ABB RobotStudio station: kostka_final.rspag

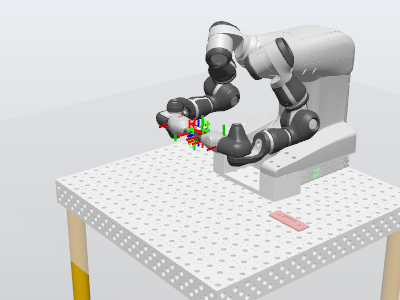
--- station ---
Station kostka (saved by RobotStudio 24.1.10693.0)
Controller Controller1
  mechanical unit ROB_R: IRB14000_0.5_0.5_R, 6 joints, base frame (0, 0, 0) mm
  mechanical unit ROB_R_7: IRB14000_0.5_0.5_R, 1 joints, base frame (0, 0, 0) mm
  mechanical unit ROB_L: IRB14000_0.5_0.5_L, 6 joints, base frame (0, 0, 0) mm
  mechanical unit ROB_L_7: IRB14000_0.5_0.5_L, 1 joints, base frame (0, 0, 0) mm
Layout (positions relative to the parent item):
  - Workplace [part, from Components\Table_for_yumi.rslib] at (-401.98, -347.06, -251) mm
  - IRB14000_0.5_0.5 [mechanism, from %ABB.RobotStudio.Models.IRB14000%\IRB14000_0.5_0.5__02.rslib] at (0, 0, 0) mm
  - IRB14000_0.5_0.5_R [mechanism, from %ABB.RobotStudio.Models.IRB14000%\IRB14000_0.5_0.5__02.rslib] at (0, 0, 0) mm; joint values [1.5163, -2.3974, -0.8514, 0.598, -1.3187, 1.4925, 3.1384] (rad or m)
  - IRB14000_0.5_0.5_L [mechanism, from %ABB.RobotStudio.Models.IRB14000%\IRB14000_0.5_0.5__02.rslib] at (0, 0, 0) mm; joint values [-1.536, -2.4067, 0.8768, 0.6099, 1.3554, 1.4655, 3.1349] (rad or m)
  - Smart_Gripper_Servo_Fingers_R [mechanism] at (341.28, 130.02, 173.54) mm, rotated rx 90 ry 0 rz 0 deg; joint values [0.023] (rad or m)
      TCP Servo at (0, 0, 114.2) mm
      links: HandBase, DownFinger, UpFinger, VacuumOne, VacuumTwo
  - Smart_Gripper_Servo_Fingers_2L [mechanism] at (341.28, -144.48, 173.54) mm, rotated rx -90 ry 0 rz 0 deg; joint values [0.023] (rad or m)
      TCP Servo at (0, 0, 114.2) mm
      links: HandBase, DownFinger, UpFinger, VacuumOne, VacuumTwo
  - Node1_con [part] at (329.77, -18.73, 185.04) mm, size 23 x 23 x 23 mm
  - Node2_con [part] at (329.77, 4.27, 162.04) mm, size 23 x 23 x 23 mm
  - Node3_con [part] at (352.77, 4.27, 162.04) mm, size 23 x 23 x 23 mm
  - Node4_con [part] at (329.78, -18.73, 162.04) mm, size 23 x 23 x 23 mm
  - Node5_con [part] at (352.77, -18.73, 162.04) mm, size 23 x 23 x 23 mm
  - Node6_con [part] at (352.77, 4.27, 185.04) mm, size 23 x 23 x 23 mm
  - Node7_con [part] at (329.77, 4.27, 185.04) mm, size 23 x 23 x 23 mm
  - Node8_con [part] at (352.77, -18.73, 185.04) mm, size 23 x 23 x 23 mm
  - Positioner [smart component, from Components\Positioner.rslib]
      properties: Object=Node1_con; Position=[0.329775 -0.01873 0.185036]; Orientation=[0 0 0]; Reference=Global; ReferenceObject=(none)
  - Positioner_2 [smart component, from Components\Positioner.rslib]
      properties: Object=Node2_con; Position=[0.329775 0.00427 0.162037]; Orientation=[0 0 0]; Reference=Global; ReferenceObject=(none)
  - Positioner_3 [smart component, from Components\Positioner.rslib]
      properties: Object=Node3_con; Position=[0.352771 0.00427 0.162036]; Orientation=[0 0 0]; Reference=Global; ReferenceObject=(none)
  - Positioner_4 [smart component, from Components\Positioner.rslib]
      properties: Object=Node4_con; Position=[0.329775 -0.01873 0.162037]; Orientation=[0 0 0]; Reference=Global; ReferenceObject=(none)
  - Positioner_5 [smart component, from Components\Positioner.rslib]
      properties: Object=Node5_con; Position=[0.352771 -0.01873 0.162036]; Orientation=[0 0 0]; Reference=Global; ReferenceObject=(none)
  - Positioner_6 [smart component, from Components\Positioner.rslib]
      properties: Object=Node6_con; Position=[0.352771 0.00427 0.185036]; Orientation=[0 0 0]; Reference=Global; ReferenceObject=(none)
  - Positioner_7 [smart component, from Components\Positioner.rslib]
      properties: Object=Node7_con; Position=[0.329775 0.00427 0.185036]; Orientation=[0 0 0]; Reference=Global; ReferenceObject=(none)
  - Positioner_8 [smart component, from Components\Positioner.rslib]
      properties: Object=Node8_con; Position=[0.352771 -0.01873 0.185036]; Orientation=[0 0 0]; Reference=Global; ReferenceObject=(none)
Attachment: Smart_Gripper_Servo_Fingers_R is attached to IRB14000_0.5_0.5_L / Link7
Attachment: Smart_Gripper_Servo_Fingers_2L is attached to IRB14000_0.5_0.5_R / Link7
Attachment: Node6_con is attached to Smart_Gripper_Servo_Fingers_R / HandBase
Attachment: Node7_con is attached to Smart_Gripper_Servo_Fingers_R / HandBase
Attachment: Node3_con is attached to Smart_Gripper_Servo_Fingers_R / HandBase
Attachment: Node2_con is attached to Smart_Gripper_Servo_Fingers_R / HandBase
Attachment: Node8_con is attached to Smart_Gripper_Servo_Fingers_2L / HandBase
Attachment: Node1_con is attached to Smart_Gripper_Servo_Fingers_2L / HandBase
Attachment: Node4_con is attached to Smart_Gripper_Servo_Fingers_2L / HandBase
Attachment: Node5_con is attached to Smart_Gripper_Servo_Fingers_2L / HandBase
EventTableEntry 7537: ActivationMode=2, Cyclic=false, Group=, Trigger=DO_ATTACH_1_GL 7538, Actions=[EventTableActionAttach 7572, EventTableActionAttach 7573, EventTableActionAttach 7574, EventTableActionAttach 7575], Comment=
EventTableTriggerIO 7538: Operator=0, IOValue=[1], IRC5Controller=? -1, SignalSource=Controller1 3578
EventTableEntry 7543: ActivationMode=2, Cyclic=false, Group=, Trigger=DO_DETACH_GL 7544, Actions=[EventTableActionDetach 7545], Comment=
EventTableTriggerIO 7544: Operator=0, IOValue=[1], IRC5Controller=? -1, SignalSource=Controller1 3578
EventTableActionDetach 7545: AttachmentParent=Smart_Gripper_Servo_Fingers_2L 3564, AttachmentChild=? -1
EventTableTriggerIO 7564: Operator=0, IOValue=[1], IRC5Controller=? -1, SignalSource=Controller1 3578
EventTableTriggerIO 7565: Operator=0, IOValue=[1], IRC5Controller=? -1, SignalSource=Controller1 3578
EventTableTriggerIO 7566: Operator=0, IOValue=[1], IRC5Controller=? -1, SignalSource=Controller1 3578
EventTableTriggerIO 7567: Operator=0, IOValue=[1], IRC5Controller=? -1, SignalSource=Controller1 3578
EventTableTriggerIO 7568: Operator=0, IOValue=[1], IRC5Controller=? -1, SignalSource=Controller1 3578
EventTableTriggerIO 7569: Operator=0, IOValue=[1], IRC5Controller=? -1, SignalSource=Controller1 3578
EventTableTriggerIO 7570: Operator=0, IOValue=[1], IRC5Controller=? -1, SignalSource=Controller1 3578
EventTableTriggerIO 7571: Operator=0, IOValue=[1], IRC5Controller=? -1, SignalSource=Controller1 3578
EventTableActionAttach 7572: MountObject=false, FlangeIndext=0, FindNearest=false, AttachmentParent=Smart_Gripper_Servo_Fingers_2L 3564, AttachmentChild=Node8_con 7749, Offset=[X=1, Y=0, Z=0, W=0, X=0, Y=1, Z=0, W=0, X=0, Y=0, Z=1, W=0, X=0, Y=0, Z=0, W=1]
EventTableActionAttach 7573: MountObject=false, FlangeIndext=0, FindNearest=false, AttachmentParent=Smart_Gripper_Servo_Fingers_2L 3564, AttachmentChild=Node6_con 7745, Offset=[X=1, Y=0, Z=0, W=0, X=0, Y=1, Z=0, W=0, X=0, Y=0, Z=1, W=0, X=0, Y=0, Z=0, W=1]
EventTableActionAttach 7574: MountObject=false, FlangeIndext=0, FindNearest=false, AttachmentParent=Smart_Gripper_Servo_Fingers_2L 3564, AttachmentChild=Node5_con 7743, Offset=[X=1, Y=0, Z=0, W=0, X=0, Y=1, Z=0, W=0, X=0, Y=0, Z=1, W=0, X=0, Y=0, Z=0, W=1]
EventTableActionAttach 7575: MountObject=false, FlangeIndext=0, FindNearest=false, AttachmentParent=Smart_Gripper_Servo_Fingers_2L 3564, AttachmentChild=Node3_con 7739, Offset=[X=1, Y=0, Z=0, W=0, X=0, Y=1, Z=0, W=0, X=0, Y=0, Z=1, W=0, X=0, Y=0, Z=0, W=1]
EventTableTriggerIO 7576: Operator=0, IOValue=[1], IRC5Controller=? -1, SignalSource=Controller1 3578
EventTableEntry 7577: ActivationMode=2, Cyclic=false, Group=, Trigger=DO_ATTACH_2_GL 7564, Actions=[EventTableActionAttach 7578, EventTableActionAttach 7579, EventTableActionAttach 7580, EventTableActionAttach 7581], Comment=
EventTableActionAttach 7578: MountObject=false, FlangeIndext=0, FindNearest=false, AttachmentParent=Smart_Gripper_Servo_Fingers_2L 3564, AttachmentChild=Node8_con 7749, Offset=[X=1, Y=0, Z=0, W=0, X=0, Y=1, Z=0, W=0, X=0, Y=0, Z=1, W=0, X=0, Y=0, Z=0, W=1]
EventTableActionAttach 7579: MountObject=false, FlangeIndext=0, FindNearest=false, AttachmentParent=Smart_Gripper_Servo_Fingers_2L 3564, AttachmentChild=Node1_con 7735, Offset=[X=1, Y=0, Z=0, W=0, X=0, Y=1, Z=0, W=0, X=0, Y=0, Z=1, W=0, X=0, Y=0, Z=0, W=1]
EventTableActionAttach 7580: MountObject=false, FlangeIndext=0, FindNearest=false, AttachmentParent=Smart_Gripper_Servo_Fingers_2L 3564, AttachmentChild=Node4_con 7741, Offset=[X=1, Y=0, Z=0, W=0, X=0, Y=1, Z=0, W=0, X=0, Y=0, Z=1, W=0, X=0, Y=0, Z=0, W=1]
EventTableActionAttach 7581: MountObject=false, FlangeIndext=0, FindNearest=false, AttachmentParent=Smart_Gripper_Servo_Fingers_2L 3564, AttachmentChild=Node5_con 7743, Offset=[X=1, Y=0, Z=0, W=0, X=0, Y=1, Z=0, W=0, X=0, Y=0, Z=1, W=0, X=0, Y=0, Z=0, W=1]
EventTableEntry 7582: ActivationMode=2, Cyclic=false, Group=, Trigger=DO_ATTACH_5_GR 7568, Actions=[EventTableActionAttach 7583, EventTableActionAttach 7584, EventTableActionAttach 7585, EventTableActionAttach 7586], Comment=
EventTableActionAttach 7583: MountObject=false, FlangeIndext=0, FindNearest=false, AttachmentParent=Smart_Gripper_Servo_Fingers_R 3556, AttachmentChild=Node1_con 7735, Offset=[X=1, Y=0, Z=0, W=0, X=0, Y=1, Z=0, W=0, X=0, Y=0, Z=1, W=0, X=0, Y=0, Z=0, W=1]
EventTableActionAttach 7584: MountObject=false, FlangeIndext=0, FindNearest=false, AttachmentParent=Smart_Gripper_Servo_Fingers_R 3556, AttachmentChild=Node2_con 7737, Offset=[X=1, Y=0, Z=0, W=0, X=0, Y=1, Z=0, W=0, X=0, Y=0, Z=1, W=0, X=0, Y=0, Z=0, W=1]
EventTableActionAttach 7585: MountObject=false, FlangeIndext=0, FindNearest=false, AttachmentParent=Smart_Gripper_Servo_Fingers_R 3556, AttachmentChild=Node7_con 7747, Offset=[X=1, Y=0, Z=0, W=0, X=0, Y=1, Z=0, W=0, X=0, Y=0, Z=1, W=0, X=0, Y=0, Z=0, W=1]
EventTableActionAttach 7586: MountObject=false, FlangeIndext=0, FindNearest=false, AttachmentParent=Smart_Gripper_Servo_Fingers_R 3556, AttachmentChild=Node4_con 7741, Offset=[X=1, Y=0, Z=0, W=0, X=0, Y=1, Z=0, W=0, X=0, Y=0, Z=1, W=0, X=0, Y=0, Z=0, W=1]
EventTableEntry 7587: ActivationMode=2, Cyclic=false, Group=, Trigger=DO_DETACH_GR 7576, Actions=[EventTableActionDetach 7588], Comment=
EventTableActionDetach 7588: AttachmentParent=Smart_Gripper_Servo_Fingers_R 3556, AttachmentChild=? -1
EventTableEntry 7589: ActivationMode=2, Cyclic=false, Group=, Trigger=DO_ATTACH_4_GR 7569, Actions=[EventTableActionAttach 7590, EventTableActionAttach 7591, EventTableActionAttach 7592, EventTableActionAttach 7593], Comment=
EventTableActionAttach 7590: MountObject=false, FlangeIndext=0, FindNearest=false, AttachmentParent=Smart_Gripper_Servo_Fingers_R 3556, AttachmentChild=Node6_con 7745, Offset=[X=1, Y=0, Z=0, W=0, X=0, Y=1, Z=0, W=0, X=0, Y=0, Z=1, W=0, X=0, Y=0, Z=0, W=1]
EventTableActionAttach 7591: MountObject=false, FlangeIndext=0, FindNearest=false, AttachmentParent=Smart_Gripper_Servo_Fingers_R 3556, AttachmentChild=Node7_con 7747, Offset=[X=1, Y=0, Z=0, W=0, X=0, Y=1, Z=0, W=0, X=0, Y=0, Z=1, W=0, X=0, Y=0, Z=0, W=1]
EventTableActionAttach 7592: MountObject=false, FlangeIndext=0, FindNearest=false, AttachmentParent=Smart_Gripper_Servo_Fingers_R 3556, AttachmentChild=Node3_con 7739, Offset=[X=1, Y=0, Z=0, W=0, X=0, Y=1, Z=0, W=0, X=0, Y=0, Z=1, W=0, X=0, Y=0, Z=0, W=1]
EventTableActionAttach 7593: MountObject=false, FlangeIndext=0, FindNearest=false, AttachmentParent=Smart_Gripper_Servo_Fingers_R 3556, AttachmentChild=Node2_con 7737, Offset=[X=1, Y=0, Z=0, W=0, X=0, Y=1, Z=0, W=0, X=0, Y=0, Z=1, W=0, X=0, Y=0, Z=0, W=1]
EventTableEntry 7594: ActivationMode=2, Cyclic=false, Group=, Trigger=DO_ATTACH_3_GR 7570, Actions=[EventTableActionAttach 7595, EventTableActionAttach 7596, EventTableActionAttach 7597, EventTableActionAttach 7598], Comment=
EventTableActionAttach 7595: MountObject=false, FlangeIndext=0, FindNearest=false, AttachmentParent=Smart_Gripper_Servo_Fingers_R 3556, AttachmentChild=Node2_con 7737, Offset=[X=1, Y=0, Z=0, W=0, X=0, Y=1, Z=0, W=0, X=0, Y=0, Z=1, W=0, X=0, Y=0, Z=0, W=1]
EventTableActionAttach 7596: MountObject=false, FlangeIndext=0, FindNearest=false, AttachmentParent=Smart_Gripper_Servo_Fingers_R 3556, AttachmentChild=Node3_con 7739, Offset=[X=1, Y=0, Z=0, W=0, X=0, Y=1, Z=0, W=0, X=0, Y=0, Z=1, W=0, X=0, Y=0, Z=0, W=1]
EventTableActionAttach 7597: MountObject=false, FlangeIndext=0, FindNearest=false, AttachmentParent=Smart_Gripper_Servo_Fingers_R 3556, AttachmentChild=Node4_con 7741, Offset=[X=1, Y=0, Z=0, W=0, X=0, Y=1, Z=0, W=0, X=0, Y=0, Z=1, W=0, X=0, Y=0, Z=0, W=1]
EventTableActionAttach 7598: MountObject=false, FlangeIndext=0, FindNearest=false, AttachmentParent=Smart_Gripper_Servo_Fingers_R 3556, AttachmentChild=Node5_con 7743, Offset=[X=1, Y=0, Z=0, W=0, X=0, Y=1, Z=0, W=0, X=0, Y=0, Z=1, W=0, X=0, Y=0, Z=0, W=1]
EventTableEntry 7599: ActivationMode=2, Cyclic=false, Group=, Trigger=DO_ATTACH_6_GL 7571, Actions=[EventTableActionAttach 7600, EventTableActionAttach 7601, EventTableActionAttach 7602, EventTableActionAttach 7603], Comment=
EventTableActionAttach 7600: MountObject=false, FlangeIndext=0, FindNearest=false, AttachmentParent=Smart_Gripper_Servo_Fingers_2L 3564, AttachmentChild=Node1_con 7735, Offset=[X=1, Y=0, Z=0, W=0, X=0, Y=1, Z=0, W=0, X=0, Y=0, Z=1, W=0, X=0, Y=0, Z=0, W=1]
EventTableActionAttach 7601: MountObject=false, FlangeIndext=0, FindNearest=false, AttachmentParent=Smart_Gripper_Servo_Fingers_2L 3564, AttachmentChild=Node8_con 7749, Offset=[X=1, Y=0, Z=0, W=0, X=0, Y=1, Z=0, W=0, X=0, Y=0, Z=1, W=0, X=0, Y=0, Z=0, W=1]
EventTableActionAttach 7602: MountObject=false, FlangeIndext=0, FindNearest=false, AttachmentParent=Smart_Gripper_Servo_Fingers_2L 3564, AttachmentChild=Node7_con 7747, Offset=[X=1, Y=0, Z=0, W=0, X=0, Y=1, Z=0, W=0, X=0, Y=0, Z=1, W=0, X=0, Y=0, Z=0, W=1]
EventTableActionAttach 7603: MountObject=false, FlangeIndext=0, FindNearest=false, AttachmentParent=Smart_Gripper_Servo_Fingers_2L 3564, AttachmentChild=Node6_con 7745, Offset=[X=1, Y=0, Z=0, W=0, X=0, Y=1, Z=0, W=0, X=0, Y=0, Z=1, W=0, X=0, Y=0, Z=0, W=1]
EventTableEntry 7630: ActivationMode=2, Cyclic=false, Group=, Trigger=DO_CLOSE_GL 7631, Actions=[EventTableActionMechanicalPose 7632], Comment=
EventTableTriggerIO 7631: Operator=0, IOValue=[1], IRC5Controller=? -1, SignalSource=Controller1 3578
EventTableActionMechanicalPose 7632: VirtualSignal=, Mechanism=Smart_Gripper_Servo_Fingers_2L 3564, ToPoseName=SyncPosition, VirtualSignalValue=[1]
EventTableTriggerIO 7633: Operator=0, IOValue=[1], IRC5Controller=? -1, SignalSource=Controller1 3578
EventTableTriggerIO 7634: Operator=0, IOValue=[1], IRC5Controller=? -1, SignalSource=Controller1 3578
EventTableTriggerIO 7635: Operator=0, IOValue=[1], IRC5Controller=? -1, SignalSource=Controller1 3578
EventTableEntry 7636: ActivationMode=2, Cyclic=false, Group=, Trigger=DO_OPEN_GL 7633, Actions=[EventTableActionMechanicalPose 7637], Comment=
EventTableActionMechanicalPose 7637: VirtualSignal=, Mechanism=Smart_Gripper_Servo_Fingers_2L 3564, ToPoseName=HomePosition, VirtualSignalValue=[1]
EventTableEntry 7638: ActivationMode=2, Cyclic=false, Group=, Trigger=DO_CLOSE_GR 7634, Actions=[EventTableActionMechanicalPose 7639], Comment=
EventTableActionMechanicalPose 7639: VirtualSignal=, Mechanism=Smart_Gripper_Servo_Fingers_R 3556, ToPoseName=SyncPosition, VirtualSignalValue=[1]
EventTableEntry 7640: ActivationMode=2, Cyclic=false, Group=, Trigger=DO_OPEN_GR 7635, Actions=[EventTableActionMechanicalPose 7641], Comment=
EventTableActionMechanicalPose 7641: VirtualSignal=, Mechanism=Smart_Gripper_Servo_Fingers_R 3556, ToPoseName=HomePosition, VirtualSignalValue=[1]
EventTableTriggerIO 7692: Operator=0, IOValue=[1], IRC5Controller=? -1, SignalSource=Controller1 3578
EventTableTriggerIO 7693: Operator=0, IOValue=[1], IRC5Controller=? -1, SignalSource=Controller1 3578
EventTableTriggerIO 7694: Operator=0, IOValue=[1], IRC5Controller=? -1, SignalSource=Controller1 3578
EventTableTriggerIO 7695: Operator=0, IOValue=[1], IRC5Controller=? -1, SignalSource=Controller1 3578
EventTableTriggerIO 7696: Operator=0, IOValue=[1], IRC5Controller=? -1, SignalSource=Controller1 3578
EventTableTriggerIO 7697: Operator=0, IOValue=[1], IRC5Controller=? -1, SignalSource=Controller1 3578
EventTableTriggerIO 7698: Operator=0, IOValue=[1], IRC5Controller=? -1, SignalSource=Controller1 3578
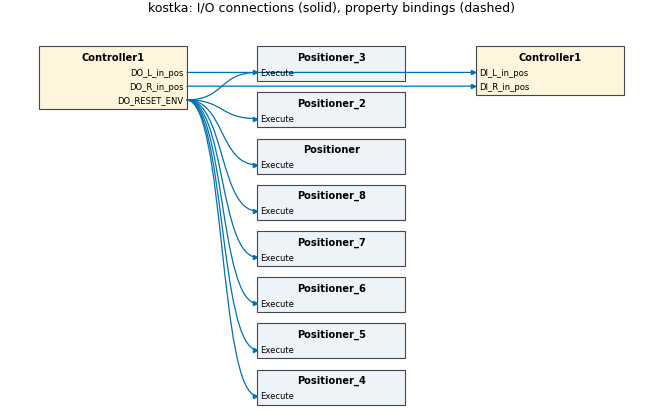
Station logic (signal -> signal, property => property):
  Controller1.DO_L_in_pos -> Controller1.DI_L_in_pos
  Controller1.DO_R_in_pos -> Controller1.DI_R_in_pos
  Controller1.DO_RESET_ENV -> Positioner_3.Execute
  Controller1.DO_RESET_ENV -> Positioner_2.Execute
  Controller1.DO_RESET_ENV -> Positioner.Execute
  Controller1.DO_RESET_ENV -> Positioner_8.Execute
  Controller1.DO_RESET_ENV -> Positioner_7.Execute
  Controller1.DO_RESET_ENV -> Positioner_6.Execute
  Controller1.DO_RESET_ENV -> Positioner_5.Execute
  Controller1.DO_RESET_ENV -> Positioner_4.Execute

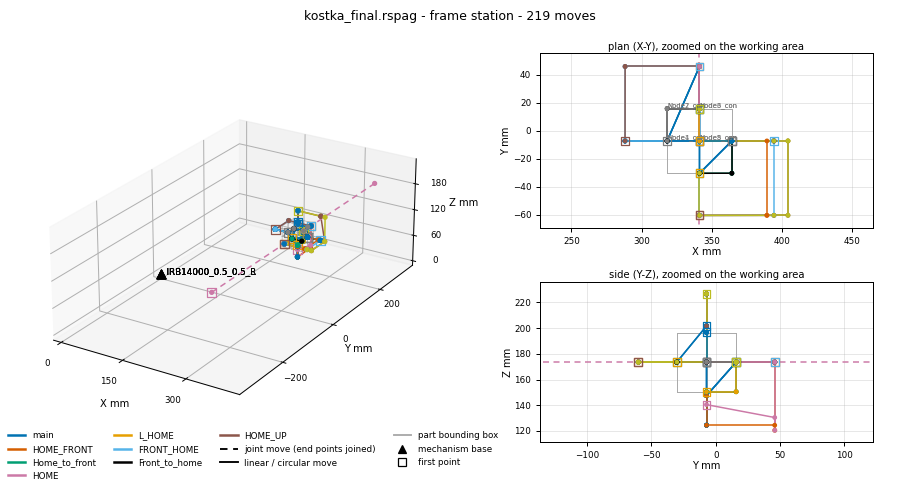
[picture p0: tool path of kostka_final.rspag in frame station, 219 of 219 moves have a stored position in this frame; points joined in program order, loops and branches not executed]
--- Controller Data/Controller1/RAPID/TASK1/PROGMOD/CalibData.mod ---
MODULE CalibData
    PERS tooldata Servo:=[TRUE,[[0,0,114.2],[1,0,0,0]],[0.215,[8.7,12.3,49.2],[1,0,0,0],0.00021,0.00024,0.00009]];
ENDMODULE

--- Controller Data/Controller1/RAPID/TASK1/PROGMOD/Module1.mod ---
MODULE Module1
        CONST robtarget Home_L:=[[341.275,-30.28,173.537],[0.707106781,-0.707106781,0,0],[1,-1,2,4],[-101.964427132,9E+09,9E+09,9E+09,9E+09,9E+09]];
    CONST robtarget Home_L_help_front:=[[364.325,-30.23,173.537],[0.707106781,-0.707106781,0,0],[1,-1,2,4],[-101.964427132,9E+09,9E+09,9E+09,9E+09,9E+09]];
    CONST robtarget L_front_help_home:=[[364.325,-30.23,173.537],[0.707106781,0,-0.707106781,0],[1,-1,2,4],[-101.96443282,9E+09,9E+09,9E+09,9E+09,9E+09]];
    CONST robtarget L_front:=[[364.325,-7.23,173.537],[0.707106781,0,-0.707106781,0],[1,-1,2,4],[-101.96443282,9E+09,9E+09,9E+09,9E+09,9E+09]];
    CONST robtarget L_front_help_up:=[[364.325,-7.23,196.537],[0.5,-0.5,-0.5,0.5],[1,-1,2,4],[-101.96443282,9E+09,9E+09,9E+09,9E+09,9E+09]];
    CONST robtarget L_up_from_front_help:=[[364.324659724,-7.23,196.536776157],[0,0,1,0],[1,-2,0,4],[-101.964427132,9E+09,9E+09,9E+09,9E+09,9E+09]];
    CONST robtarget L_up:=[[341.274659724,-7.23,196.586776157],[0,0,1,0],[1,-2,1,4],[-101.964427132,9E+09,9E+09,9E+09,9E+09,9E+09]];
    CONST robtarget L_front_ACW:=[[364.325,-7.23,173.537],[0.5,0.5,-0.5,-0.5],[1,-1,2,4],[-101.96443282,9E+09,9E+09,9E+09,9E+09,9E+09]];
    CONST robtarget L_front_CW:=[[364.325,-7.23,173.537],[0.5,-0.5,-0.5,0.5],[1,-1,-1,4],[-101.96443282,9E+09,9E+09,9E+09,9E+09,9E+09]];
    CONST robtarget Home_L_CW:=[[341.275,-30.28,173.537],[0.5,-0.5,0.5,0.5],[1,-1,2,4],[-101.964427132,9E+09,9E+09,9E+09,9E+09,9E+09]];
    CONST robtarget Home_L_ACW:=[[341.275,-30.28,173.537],[0.5,-0.5,-0.5,-0.5],[1,-1,2,4],[-101.964427132,9E+09,9E+09,9E+09,9E+09,9E+09]];
    CONST robtarget L_up_ACW:=[[341.274659724,-7.23,196.586776157],[0,-0.707106781,0.707106781,0],[1,-2,1,4],[-101.964427132,9E+09,9E+09,9E+09,9E+09,9E+09]];
    CONST robtarget L_up_CW:=[[341.274659724,-7.23,196.586776157],[0,0.707106781,0.707106781,0],[1,-2,1,4],[-101.964427132,9E+09,9E+09,9E+09,9E+09,9E+09]];

    !####################################### OBSLUHUJU U F L
    PROC main()
!        HOME;
!        MoveL Home_L_CW,v150,fine,Servo;
!        MoveL Home_L,v150,fine,Servo;
!        MoveL Home_L_ACW,v150,fine,Servo;
!        MoveL Home_L,v150,fine,Servo;
!        HOME_FRONT;
!        MoveL L_front_ACW,v150,fine,Servo;
!        MoveL L_front,v150,fine,Servo;
!        MoveL L_front_CW,v150,fine,Servo;
!        MoveL L_front,v150,fine,Servo;
!        FRONT_UP;
!        MoveL Offs(L_up_ACW,0,0,5),v150,fine,Servo;
!        MoveL Offs(L_up,0,0,5),v150,fine,Servo;
!        MoveL Offs(L_up_CW,0,0,5),v150,fine,Servo;
!        MoveL Offs(L_up,0,0,5),v150,fine,Servo;
!        UP_FRONT;
!        MoveL L_front_ACW,v150,fine,Servo;
!        MoveL L_front,v150,fine,Servo;
!        MoveL L_front_CW,v150,fine,Servo;
!        MoveL L_front,v150,fine,Servo;
!        FRONT_HOME;
!        MoveL Home_L_CW,v150,fine,Servo;
!        MoveL Home_L,v150,fine,Servo;
!        MoveL Home_L_ACW,v150,fine,Servo;
!        MoveL Home_L,v150,fine,Servo;
        VAR num SizeOfInputArray:=25;
        VAR string input_array{25};
        input_array:= ["F","F'","F2","F2","R","R'","R2","R2","U","U'","U2","U2","B","B'","B2","B2","L","L'","L2","L2","D","D'","D2","D2","BREAK"];
        !input_array:= ["U","U'","U2","U2","BREAK"];

        SetDO DO_R_in_pos,1;
        WaitDI DI_L_in_pos,1;
        WaitTime .5;
        SetDO DO_R_in_pos,0;

        PulseDO DO_OPEN_GL;
        WaitTime 5;
        HOME;
        WaitTime 10;
        PulseDO DO_CLOSE_GL;
        WaitTime 0.25;
        PulseDO DO_ATTACH_2_GL;
        WaitTime 0.25;
        SetDO DO_R_in_pos,1;
        WaitDI DI_L_in_pos,1;
        WaitTime .5;
        SetDO DO_R_in_pos,0;

      FOR i FROM 1 TO SizeOfInputArray DO
        WaitDI DI_R_in_pos,0;
        WaitDI DI_L_in_pos,0;
        TEST input_array{i}
            CASE "U" :      !cekej signal####################
                WaitDI DI_L_in_pos,1;
                PulseDO DO_OPEN_GL;
                WaitTime 0.25;
                PulseDO DO_DETACH_GL;
                WaitTime 0.25;
                HOME_UP;
                PulseDO DO_CLOSE_GL;
                WaitTime 0.25;
                PulseDO DO_ATTACH_6_GL;
                WaitTime 0.25;
                MoveL Offs(L_up_CW,0,0,5),v150,fine,Servo;
                PulseDO DO_OPEN_GL;
                WaitTime 0.25;
                PulseDO DO_DETACH_GL;
                WaitTime 0.25;
                MoveL Offs(L_up_CW,0,0,30),v150,fine,Servo;
                MoveL Offs(L_up,0,0,30),v150,fine,Servo;
                MoveL Offs(L_up,0,0,5),v150,fine,Servo;
                UP_HOME;
                PulseDO DO_CLOSE_GL;
                WaitTime 0.25;
                PulseDO DO_ATTACH_2_GL;
                WaitTime 0.25;
                SetDO DO_R_in_pos,1;
                WaitDI DI_L_in_pos,0;
                SetDO DO_R_in_pos,0;
            CASE "F" :      !cekej signal####################
                WaitDI DI_L_in_pos,1;
                PulseDO DO_OPEN_GL;
                WaitTime 0.25;
                PulseDO DO_DETACH_GL;
                WaitTime 0.25;
                HOME_FRONT;
                PulseDO DO_CLOSE_GL;
                WaitTime 0.25;
                PulseDO DO_ATTACH_1_GL;
                WaitTime 0.25;
                MoveL L_front_CW,v150,fine,Servo;
                PulseDO DO_OPEN_GL;
                WaitTime 0.25;
                PulseDO DO_DETACH_GL;
                WaitTime 0.25;
                MoveL Offs(L_front_CW,30,0,0),v150,fine,Servo;
                MoveL Offs(L_front,30,0,0),v150,fine,Servo;
                MoveL L_front,v150,fine,Servo;
                FRONT_HOME;
                PulseDO DO_CLOSE_GL;
                WaitTime 0.25;
                PulseDO DO_ATTACH_2_GL;
                WaitTime 0.25;
                SetDO DO_R_in_pos,1;
                WaitDI DI_L_in_pos,0;
                SetDO DO_R_in_pos,0;
            CASE "B" :      !NENENENEcekej signal####################
                PulseDO DO_OPEN_GL;
                WaitTime 0.25;
                PulseDO DO_DETACH_GL;
                WaitTime 0.25;
                HOME_FRONT;
                PulseDO DO_CLOSE_GL;
                WaitTime 0.25;
                PulseDO DO_ATTACH_1_GL;
                WaitTime 0.25;
                SetDO DO_R_in_pos,1;
                WaitDI DI_L_in_pos,1;
                PulseDO DO_OPEN_GL;
                WaitTime 0.25;
                PulseDO DO_DETACH_GL;
                WaitTime 0.25;
                FRONT_HOME;
                PulseDO DO_CLOSE_GL;
                WaitTime 0.25;
                PulseDO DO_ATTACH_2_GL;
                WaitTime 0.25;
                SetDO DO_R_in_pos,0;
            CASE "L" :      !cekej signal####################
!                WaitDI DI_L_in_pos,1;
!                PulseDO DO_OPEN_GL;
!                HOME;
!                PulseDO DO_CLOSE_GL;
                MoveL Home_L_CW,v150,fine,Servo;
                PulseDO DO_OPEN_GL;
                WaitTime 0.25;
                PulseDO DO_DETACH_GL;
                WaitTime 0.25;
                MoveL Offs(Home_L_CW,0,-30,0),v150,fine,Servo;
                MoveL Offs(Home_L,0,-30,0),v150,fine,Servo;
                MoveL Home_L,v150,fine,Servo;
!                HOME;
                PulseDO DO_CLOSE_GL;
                WaitTime 0.25;
                PulseDO DO_ATTACH_2_GL;
                WaitTime 0.25;
!                SetDO DO_R_in_pos,1;
!                WaitDI DI_L_in_pos,0;
!                SetDO DO_R_in_pos,0;
            CASE "R" :      !NENENENEcekej signal####################
!                PulseDO DO_OPEN_GL;
!                HOME;
!                PulseDO DO_CLOSE_GL;
!                SetDO DO_R_in_pos,1;
!                WaitDI DI_L_in_pos,1;
!                PulseDO DO_OPEN_GL;
!                HOME;
!                PulseDO DO_CLOSE_GL;
!                SetDO DO_R_in_pos,0;
            CASE "D" :      !NENENENEcekej signal####################
                PulseDO DO_OPEN_GL;
                WaitTime 0.25;
                PulseDO DO_DETACH_GL;
                WaitTime 0.25;
                HOME_UP;
                PulseDO DO_CLOSE_GL;
                WaitTime 0.25;
                PulseDO DO_ATTACH_6_GL;
                WaitTime 0.25;
                SetDO DO_R_in_pos,1;
                WaitDI DI_L_in_pos,1;
                PulseDO DO_OPEN_GL;
                WaitTime 0.25;
                PulseDO DO_DETACH_GL;
                WaitTime 0.25;
                UP_HOME;
                PulseDO DO_CLOSE_GL;
                WaitTime 0.25;
                PulseDO DO_ATTACH_2_GL;
                WaitTime 0.25;
                SetDO DO_R_in_pos,0;
            CASE "U2" :
                WaitDI DI_L_in_pos,1;
                PulseDO DO_OPEN_GL;
                WaitTime 0.25;
                PulseDO DO_DETACH_GL;
                WaitTime 0.25;
                HOME_UP;
                PulseDO DO_CLOSE_GL;
                WaitTime 0.25;
                PulseDO DO_ATTACH_6_GL;
                WaitTime 0.25;
                MoveL Offs(L_up_CW,0,0,5),v150,fine,Servo;
                PulseDO DO_OPEN_GL;
                WaitTime 0.25;
                PulseDO DO_DETACH_GL;
                WaitTime 0.25;
                MoveL Offs(L_up_CW,0,0,30),v150,fine,Servo;
                MoveL Offs(L_up,0,0,30),v150,fine,Servo;
                MoveL Offs(L_up,0,0,5),v150,fine,Servo;
                PulseDO DO_CLOSE_GL;
                WaitTime 0.25;
                PulseDO DO_ATTACH_6_GL;
                WaitTime 0.25;
                MoveL Offs(L_up_CW,0,0,5),v150,fine,Servo;
                PulseDO DO_OPEN_GL;
                WaitTime 0.25;
                PulseDO DO_DETACH_GL;
                WaitTime 0.25;
                MoveL Offs(L_up_CW,0,0,30),v150,fine,Servo;
                MoveL Offs(L_up,0,0,30),v150,fine,Servo;
                MoveL Offs(L_up,0,0,5),v150,fine,Servo;
                UP_HOME;
                PulseDO DO_CLOSE_GL;
                WaitTime 0.25;
                PulseDO DO_ATTACH_2_GL;
                WaitTime 0.25;
                SetDO DO_R_in_pos,1;
                WaitDI DI_L_in_pos,0;
                SetDO DO_R_in_pos,0;
            CASE "F2" :
                WaitDI DI_L_in_pos,1;
                PulseDO DO_OPEN_GL;
                WaitTime 0.25;
                PulseDO DO_DETACH_GL;
                WaitTime 0.25;
                HOME_FRONT;
                PulseDO DO_CLOSE_GL;
                WaitTime 0.25;
                PulseDO DO_ATTACH_1_GL;
                WaitTime 0.25;
                MoveL L_front_CW,v150,fine,Servo;
                PulseDO DO_OPEN_GL;
                WaitTime 0.25;
                PulseDO DO_DETACH_GL;
                WaitTime 0.25;
                MoveL Offs(L_front_CW,30,0,0),v150,fine,Servo;
                MoveL Offs(L_front,30,0,0),v150,fine,Servo;
                MoveL L_front,v150,fine,Servo;
                PulseDO DO_CLOSE_GL;
                WaitTime 0.25;
                PulseDO DO_ATTACH_1_GL;
                WaitTime 0.25;
                MoveL L_front_CW,v150,fine,Servo;
                PulseDO DO_OPEN_GL;
                WaitTime 0.25;
                PulseDO DO_DETACH_GL;
                WaitTime 0.25;
                MoveL Offs(L_front_CW,30,0,0),v150,fine,Servo;
                MoveL Offs(L_front,30,0,0),v150,fine,Servo;
                MoveL L_front,v150,fine,Servo;
                FRONT_HOME;
                PulseDO DO_CLOSE_GL;
                WaitTime 0.25;
                PulseDO DO_ATTACH_2_GL;
                WaitTime 0.25;
                SetDO DO_R_in_pos,1;
                WaitDI DI_L_in_pos,0;
                SetDO DO_R_in_pos,0;
            CASE "B2" :
                PulseDO DO_OPEN_GL;
                WaitTime 0.25;
                PulseDO DO_DETACH_GL;
                WaitTime 0.25;
                HOME_FRONT;
                PulseDO DO_CLOSE_GL;
                WaitTime 0.25;
                PulseDO DO_ATTACH_1_GL;
                WaitTime 0.25;
                SetDO DO_R_in_pos,1;
                WaitDI DI_L_in_pos,1;
                PulseDO DO_OPEN_GL;
                WaitTime 0.25;
                PulseDO DO_DETACH_GL;
                WaitTime 0.25;
                FRONT_HOME;
                PulseDO DO_CLOSE_GL;
                WaitTime 0.25;
                PulseDO DO_ATTACH_2_GL;
                WaitTime 0.25;
                SetDO DO_R_in_pos,0;
            CASE "L2" :
!                WaitDI DI_L_in_pos,1;
!                PulseDO DO_OPEN_GL;
!                HOME;
!                PulseDO DO_CLOSE_GL;
                MoveL Home_L_CW,v150,fine,Servo;
                PulseDO DO_OPEN_GL;
                WaitTime 0.25;
                PulseDO DO_DETACH_GL;
                WaitTime 0.25;
                MoveL Offs(Home_L_CW,0,-30,0),v150,fine,Servo;
                MoveL Offs(Home_L,0,-30,0),v150,fine,Servo;
                MoveL Home_L,v150,fine,Servo;
!                HOME;
                PulseDO DO_CLOSE_GL;
                WaitTime 0.25;
                PulseDO DO_ATTACH_2_GL;
                WaitTime 0.25;
                MoveL Home_L_CW,v150,fine,Servo;
                PulseDO DO_OPEN_GL;
                WaitTime 0.25;
                PulseDO DO_DETACH_GL;
                WaitTime 0.25;
                MoveL Offs(Home_L_CW,0,-30,0),v150,fine,Servo;
                MoveL Offs(Home_L,0,-30,0),v150,fine,Servo;
                MoveL Home_L,v150,fine,Servo;
!                HOME;
                PulseDO DO_CLOSE_GL;
                WaitTime 0.25;
                PulseDO DO_ATTACH_2_GL;
                WaitTime 0.25;
!                SetDO DO_R_in_pos,1;
!                WaitDI DI_L_in_pos,0;
!                SetDO DO_R_in_pos,0;
            CASE "R2" :
!                PulseDO DO_OPEN_GL;
!                HOME;
!                PulseDO DO_CLOSE_GL;
!                SetDO DO_R_in_pos,1;
!                WaitDI DI_L_in_pos,1;
!                PulseDO DO_OPEN_GL;
!                HOME;
!                PulseDO DO_CLOSE_GL;
!                SetDO DO_R_in_pos,0;
            CASE "D2" :
                PulseDO DO_OPEN_GL;
                WaitTime 0.25;
                PulseDO DO_DETACH_GL;
                WaitTime 0.25;
                HOME_UP;
                PulseDO DO_CLOSE_GL;
                WaitTime 0.25;
                PulseDO DO_ATTACH_6_GL;
                WaitTime 0.25;
                SetDO DO_R_in_pos,1;
                WaitDI DI_L_in_pos,1;
                PulseDO DO_OPEN_GL;
                WaitTime 0.25;
                PulseDO DO_DETACH_GL;
                WaitTime 0.25;
                UP_HOME;
                PulseDO DO_CLOSE_GL;
                WaitTime 0.25;
                PulseDO DO_ATTACH_2_GL;
                WaitTime 0.25;
                SetDO DO_R_in_pos,0;
            CASE "U'" :
                WaitDI DI_L_in_pos,1;
                PulseDO DO_OPEN_GL;
                WaitTime 0.25;
                PulseDO DO_DETACH_GL;
                WaitTime 0.25;
                HOME_UP;
                PulseDO DO_CLOSE_GL;
                WaitTime 0.25;
                PulseDO DO_ATTACH_6_GL;
                WaitTime 0.25;
                MoveL Offs(L_up_ACW,0,0,5),v150,fine,Servo;
                PulseDO DO_OPEN_GL;
                WaitTime 0.25;
                PulseDO DO_DETACH_GL;
                WaitTime 0.25;
                MoveL Offs(L_up_ACW,0,0,30),v150,fine,Servo;
                MoveL Offs(L_up,0,0,30),v150,fine,Servo;
                MoveL Offs(L_up,0,0,5),v150,fine,Servo;
                UP_HOME;
                PulseDO DO_CLOSE_GL;
                WaitTime 0.25;
                PulseDO DO_ATTACH_2_GL;
                WaitTime 0.25;
                SetDO DO_R_in_pos,1;
                WaitDI DI_L_in_pos,0;
                SetDO DO_R_in_pos,0;
            CASE "F'" :
                WaitDI DI_L_in_pos,1;
                PulseDO DO_OPEN_GL;
                WaitTime 0.25;
                PulseDO DO_DETACH_GL;
                WaitTime 0.25;
                HOME_FRONT;
                PulseDO DO_CLOSE_GL;
                WaitTime 0.25;
                PulseDO DO_ATTACH_1_GL;
                WaitTime 0.25;
                MoveL L_front_ACW,v150,fine,Servo;
                PulseDO DO_OPEN_GL;
                WaitTime 0.25;
                PulseDO DO_DETACH_GL;
                WaitTime 0.25;
                MoveL Offs(L_front_ACW,30,0,0),v150,fine,Servo;
                MoveL Offs(L_front,30,0,0),v150,fine,Servo;
                MoveL L_front,v150,fine,Servo;
                FRONT_HOME;
                PulseDO DO_CLOSE_GL;
                WaitTime 0.25;
                PulseDO DO_ATTACH_2_GL;
                WaitTime 0.25;
                SetDO DO_R_in_pos,1;
                WaitDI DI_L_in_pos,0;
                SetDO DO_R_in_pos,0;
            CASE "B'" :
                PulseDO DO_OPEN_GL;
                WaitTime 0.25;
                PulseDO DO_DETACH_GL;
                WaitTime 0.25;
                HOME_FRONT;
                PulseDO DO_CLOSE_GL;
                WaitTime 0.25;
                PulseDO DO_ATTACH_1_GL;
                WaitTime 0.25;
                SetDO DO_R_in_pos,1;
                WaitDI DI_L_in_pos,1;
                PulseDO DO_OPEN_GL;
                WaitTime 0.25;
                PulseDO DO_DETACH_GL;
                WaitTime 0.25;
                FRONT_HOME;
                PulseDO DO_CLOSE_GL;
                WaitTime 0.25;
                PulseDO DO_ATTACH_2_GL;
                WaitTime 0.25;
                SetDO DO_R_in_pos,0;
            CASE "L'" :
!                WaitDI DI_L_in_pos,1;
!                PulseDO DO_OPEN_GL;
!                HOME;
!                PulseDO DO_CLOSE_GL;
                MoveL Home_L_ACW,v150,fine,Servo;
                PulseDO DO_OPEN_GL;
                WaitTime 0.25;
                PulseDO DO_DETACH_GL;
                WaitTime 0.25;
                MoveL Offs(Home_L_ACW,0,-30,0),v150,fine,Servo;
                MoveL Offs(Home_L,0,-30,0),v150,fine,Servo;
                MoveL Home_L,v150,fine,Servo;
!                HOME;
                PulseDO DO_CLOSE_GL;
                WaitTime 0.25;
                PulseDO DO_ATTACH_2_GL;
                WaitTime 0.25;
!                SetDO DO_R_in_pos,1;
!                WaitDI DI_L_in_pos,0;
!                SetDO DO_R_in_pos,0;
            CASE "R'" :
!                PulseDO DO_OPEN_GL;
!                HOME;
!                PulseDO DO_CLOSE_GL;
!                SetDO DO_R_in_pos,1;
!                WaitDI DI_L_in_pos,1;
!                PulseDO DO_OPEN_GL;
!                HOME;
!                PulseDO DO_CLOSE_GL;
!                SetDO DO_R_in_pos,0;
            CASE "D'" :
                PulseDO DO_OPEN_GL;
                WaitTime 0.25;
                PulseDO DO_DETACH_GL;
                WaitTime 0.25;
                HOME_UP;
                PulseDO DO_CLOSE_GL;
                WaitTime 0.25;
                PulseDO DO_ATTACH_6_GL;
                WaitTime 0.25;
                SetDO DO_R_in_pos,1;
                WaitDI DI_L_in_pos,1;
                PulseDO DO_OPEN_GL;
                WaitTime 0.25;
                PulseDO DO_DETACH_GL;
                WaitTime 0.25;
                UP_HOME;
                PulseDO DO_CLOSE_GL;
                WaitTime 0.25;
                PulseDO DO_ATTACH_2_GL;
                WaitTime 0.25;
                SetDO DO_R_in_pos,0;
            CASE "BREAK" :
                BREAK;
        ENDTEST

      ENDFOR

        !Add your code here
    ENDPROC
    PROC HOME_FRONT()
        MoveL Offs(Home_L,0,-30,0),v150,fine,Servo;
        MoveL Offs(Home_L_help_front,25,-30,0),v150,fine,Servo;
        MoveL Offs(L_front_help_home,25,-30,0),v150,fine,Servo;
        MoveL Offs(L_front,25,0,0),v150,fine,Servo;
        MoveL L_front,v150,fine,Servo;
    ENDPROC
    PROC Home_to_front()
        MoveL Home_L,v150,fine,Servo\WObj:=wobj0;
        MoveL Home_L_help_front,v150,fine,Servo\WObj:=wobj0;
        MoveL L_front_help_home,v150,fine,Servo\WObj:=wobj0;
        MoveL L_front,v150,fine,Servo\WObj:=wobj0;
        MoveL L_front_ACW,v150,fine,Servo\WObj:=wobj0;
        MoveL L_front,v150,fine,Servo\WObj:=wobj0;
        MoveL L_front_CW,v150,fine,Servo\WObj:=wobj0;
        MoveL L_front,v150,fine,Servo\WObj:=wobj0;
    ENDPROC
    PROC HOME()
        MoveJ Offs(Home_L,0,-300,0),v150,fine,Servo;
        MoveJ Offs(Home_L,0,-30,0),v150,fine,Servo;
        MoveL Home_L,v150,fine,Servo;
    ENDPROC
    PROC L_HOME()
        MoveJ Home_L,v150,fine,Servo\WObj:=wobj0;
        MoveL Home_L_CW,v150,fine,Servo\WObj:=wobj0;
        MoveL Home_L,v150,fine,Servo\WObj:=wobj0;
        MoveL Home_L_ACW,v150,fine,Servo\WObj:=wobj0;
        MoveL Home_L,v150,fine,Servo\WObj:=wobj0;
    ENDPROC
    PROC FRONT_HOME()
        MoveL Offs(L_front,30,0,0),v150,fine,Servo;
        MoveL Offs(L_front_help_home,30,-30,0),v150,fine,Servo;
        MoveL Offs(Home_L_help_front,30,-30,0),v150,fine,Servo;
        MoveL Offs(Home_L,0,-30,0),v150,fine,Servo;
        MoveL Home_L,v150,fine,Servo;
    ENDPROC
    PROC Front_to_home()
        MoveL L_front,v150,fine,Servo\WObj:=wobj0;
        MoveL L_front_help_home,v150,fine,Servo\WObj:=wobj0;
        MoveL Home_L_help_front,v150,fine,Servo\WObj:=wobj0;
        MoveL Home_L,v150,fine,Servo\WObj:=wobj0;
        MoveL Home_L_ACW,v150,fine,Servo\WObj:=wobj0;
        MoveL Home_L,v150,fine,Servo\WObj:=wobj0;
        MoveL Home_L_CW,v150,fine,Servo\WObj:=wobj0;
        MoveL Home_L,v150,fine,Servo\WObj:=wobj0;
    ENDPROC
    PROC HOME_UP()
        MoveL Offs(Home_L,0,-30,0),v150,fine,Servo;
        MoveL Offs(Home_L_help_front,30,-30,0),v150,fine,Servo;
        MoveL Offs(L_front_help_home,40,-30,0),v150,fine,Servo;
        MoveL Offs(L_front,40,0,0),v150,fine,Servo;
        MoveL Offs(L_front_help_up,30,0,30),v150,fine,Servo;
        MoveL Offs(L_up_from_front_help,30,0,30),v150,fine,Servo;
        MoveL Offs(L_up,0,0,30),v150,fine,Servo;
        MoveL Offs(L_up,0,0,5),v150,fine,Servo;
    ENDPROC
    PROC Front_to_up()
        MoveL L_front,v150,fine,Servo\WObj:=wobj0;
        MoveL L_front_help_up,v150,fine,Servo\WObj:=wobj0;
        MoveL L_up_from_front_help,v150,fine,Servo\WObj:=wobj0;
        MoveL L_up,v150,fine,Servo\WObj:=wobj0;
        MoveL L_up_ACW,v150,fine,Servo\WObj:=wobj0;
        MoveL L_up,v150,fine,Servo\WObj:=wobj0;
        MoveL L_up_CW,v150,fine,Servo\WObj:=wobj0;
        MoveL L_up,v150,fine,Servo\WObj:=wobj0;
    ENDPROC
    PROC UP_HOME()
        MoveL Offs(L_up,0,0,30),v150,fine,Servo;
        MoveL Offs(L_up_from_front_help,30,0,30),v150,fine,Servo;
        MoveL Offs(L_front_help_up,40,0,30),v150,fine,Servo;
        MoveL Offs(L_front,40,0,0),v150,fine,Servo;
        MoveL Offs(L_front_help_home,40,-30,0),v150,fine,Servo;
        MoveL Offs(Home_L_help_front,30,-30,0),v150,fine,Servo;
        MoveL Offs(Home_L,0,-30,0),v150,fine,Servo;
        MoveL Home_L,v150,fine,Servo;
    ENDPROC
    PROC Up_to_front()
        MoveL L_up,v150,fine,Servo\WObj:=wobj0;
        MoveL L_up_from_front_help,v150,fine,Servo\WObj:=wobj0;
        MoveL L_front_help_up,v150,fine,Servo\WObj:=wobj0;
        MoveL L_front,v150,fine,Servo\WObj:=wobj0;
        MoveL L_front_CW,v150,fine,Servo\WObj:=wobj0;
        MoveL L_front,v150,fine,Servo\WObj:=wobj0;
        MoveL L_front_ACW,v150,fine,Servo\WObj:=wobj0;
        MoveL L_front,v150,fine,Servo\WObj:=wobj0;
    ENDPROC
ENDMODULE

--- Controller Data/Controller1/RAPID/TASK2/PROGMOD/Module1.mod ---
MODULE Module1
        CONST robtarget Home_R:=[[341.274942792,15.819826991,173.537032908],[0.707106781,0.707106781,0,0],[-1,1,2,4],[101.964427132,9E+09,9E+09,9E+09,9E+09,9E+09]];
    CONST robtarget Home_R_help_down:=[[341.274942792,15.819826991,150.537032908],[0.707106781,0.707106781,0,0],[-1,1,2,4],[101.964427132,9E+09,9E+09,9E+09,9E+09,9E+09]];
    CONST robtarget R_down_help:=[[341.275429936,15.770167607,150.486370455],[1,0,0,0],[-1,0,2,4],[101.964427132,9E+09,9E+09,9E+09,9E+09,9E+09]];
    CONST robtarget R_down:=[[341.275429936,-7.229832393,150.486370455],[1,0,0,0],[-1,0,2,4],[101.964427132,9E+09,9E+09,9E+09,9E+09,9E+09]];
    CONST robtarget Home_R_help_back:=[[318.274942792,15.819826991,173.537032908],[0.707106781,0.707106781,0,0],[-1,1,2,4],[101.964427132,9E+09,9E+09,9E+09,9E+09,9E+09]];
    CONST robtarget R_back_help:=[[318.275,15.82,173.537],[0.707106781,0,0.707106781,0],[-1,-1,0,4],[101.964426744,9E+09,9E+09,9E+09,9E+09,9E+09]];
    CONST robtarget R_back:=[[318.225,-7.23,173.537],[0.707106781,0,0.707106781,0],[-1,-1,0,4],[101.964426744,9E+09,9E+09,9E+09,9E+09,9E+09]];
    CONST robtarget R_down_ACW:=[[341.275429936,-7.229832393,150.486370455],[0.707106781,0,0,-0.707106781],[-1,0,2,4],[101.964427132,9E+09,9E+09,9E+09,9E+09,9E+09]];
    CONST robtarget R_down_CW:=[[341.275429936,-7.229832393,150.486370455],[0.707106781,0,0,0.707106781],[-1,0,-1,4],[101.964427132,9E+09,9E+09,9E+09,9E+09,9E+09]];
    CONST robtarget Home_R_CW:=[[341.274942792,15.819826991,173.537032908],[0.5,0.5,-0.5,0.5],[-1,1,-1,4],[101.964427132,9E+09,9E+09,9E+09,9E+09,9E+09]];
    CONST robtarget Home_R_ACW:=[[341.274942792,15.819826991,173.537032908],[0.5,0.5,0.5,-0.5],[-1,1,2,4],[101.964427132,9E+09,9E+09,9E+09,9E+09,9E+09]];
    CONST robtarget R_back_CW:=[[318.225,-7.23,173.537],[0.5,0.5,0.5,0.5],[-1,-1,0,4],[101.964426744,9E+09,9E+09,9E+09,9E+09,9E+09]];
    CONST robtarget R_back_ACW:=[[318.225,-7.23,173.537],[0.5,-0.5,0.5,-0.5],[-1,-1,0,4],[101.964426744,9E+09,9E+09,9E+09,9E+09,9E+09]];

    !####################################### OBSLUHUJU R D B
    PROC main()

        VAR num SizeOfInputArray:=25;
        VAR string input_array{25};
        input_array:= ["F","F'","F2","F2","R","R'","R2","R2","U","U'","U2","U2","B","B'","B2","B2","L","L'","L2","L2","D","D'","D2","D2","BREAK"];
        !input_array:= ["U","U'","U2","U2","BREAK"];

        PulseDO DO_OPEN_GL;PulseDO DO_OPEN_GR;
        PulseDO DO_DETACH_GL;PulseDO DO_DETACH_GR;
        SetDO DO_L_in_pos,0;SetDO DO_R_in_pos,0;

        PulseDO DO_RESET_ENV;
        SetDO DO_L_in_pos,1;
        WaitDI DI_R_in_pos,1;
        WaitTime .5;
        SetDO DO_L_in_pos,0;

        PulseDO DO_OPEN_GR;
        WaitTime 5;
        HOME;
        WaitTime 10;
        PulseDO DO_CLOSE_GR;
        WaitTime 0.25;
        PulseDO DO_ATTACH_4_GR;
        WaitTime 0.25;
        SetDO DO_L_in_pos,1;
        WaitDI DI_R_in_pos,1;
        WaitTime .5;
        SetDO DO_L_in_pos,0;

      FOR i FROM 1 TO SizeOfInputArray DO
        WaitDI DI_R_in_pos,0;
        WaitDI DI_L_in_pos,0;
        TEST input_array{i}
            CASE "U" :      !NENENENEcekej signal####################
                PulseDO DO_OPEN_GR;
                WaitTime 0.25;
                PulseDO DO_DETACH_GR;
                WaitTime 0.25;
                HOME_DOWN;
                PulseDO DO_CLOSE_GR;
                WaitTime 0.25;
                PulseDO DO_ATTACH_3_GR;
                WaitTime 0.25;
                SetDO DO_L_in_pos,1;
                WaitDI DI_R_in_pos,1;
                PulseDO DO_OPEN_GR;
                WaitTime 0.25;
                PulseDO DO_DETACH_GR;
                WaitTime 0.25;
                DOWN_HOME;
                PulseDO DO_CLOSE_GR;
                WaitTime 0.25;
                PulseDO DO_ATTACH_4_GR;
                WaitTime 0.25;
                SetDO DO_L_in_pos,0;
            CASE "F" :      !NENENENEcekej signal####################
                PulseDO DO_OPEN_GR;
                WaitTime 0.25;
                PulseDO DO_DETACH_GR;
                WaitTime 0.25;
                HOME_BACK;
                PulseDO DO_CLOSE_GR;
                WaitTime 0.25;
                PulseDO DO_ATTACH_5_GR;
                WaitTime 0.25;
                SetDO DO_L_in_pos,1;
                WaitDI DI_R_in_pos,1;
                PulseDO DO_OPEN_GR;
                WaitTime 0.25;
                PulseDO DO_DETACH_GR;
                WaitTime 0.25;
                BACK_HOME;
                PulseDO DO_CLOSE_GR;
                WaitTime 0.25;
                PulseDO DO_ATTACH_4_GR;
                WaitTime 0.25;
                SetDO DO_L_in_pos,0;
            CASE "B" :      !cekej signal####################
                WaitDI DI_R_in_pos,1;
                PulseDO DO_OPEN_GR;
                WaitTime 0.25;
                PulseDO DO_DETACH_GR;
                WaitTime 0.25;
                HOME_BACK;
                PulseDO DO_CLOSE_GR;
                WaitTime 0.25;
                PulseDO DO_ATTACH_5_GR;
                WaitTime 0.25;
                MoveL R_back_CW,v150,fine,Servo;
                PulseDO DO_OPEN_GR;
                WaitTime 0.25;
                PulseDO DO_DETACH_GR;
                WaitTime 0.25;
                MoveL Offs(R_back_CW,-30,0,0),v150,fine,Servo;
                MoveL Offs(R_back,-30,0,0),v150,fine,Servo;
                MoveL R_back,v150,fine,Servo;
                BACK_HOME;
                PulseDO DO_CLOSE_GR;
                WaitTime 0.25;
                PulseDO DO_ATTACH_4_GR;
                WaitTime 0.25;
                SetDO DO_L_in_pos,1;
                WaitDI DI_R_in_pos,0;
                SetDO DO_L_in_pos,0;
            CASE "L" :      !NENENENEcekej signal####################   NEMELO BY BYT NIC POTREBA
!                PulseDO DO_OPEN_GR;
!                HOME;
!                PulseDO DO_CLOSE_GR;
!                SetDO DO_L_in_pos,1;
!                WaitDI DI_R_in_pos,1;
!                PulseDO DO_OPEN_GR;
!                HOME;
!                PulseDO DO_CLOSE_GR;
!                SetDO DO_L_in_pos,0;
            CASE "R" :      !cekej signal####################
!                WaitDI DI_R_in_pos,1;
!                PulseDO DO_OPEN_GR;
!                HOME;
!                PulseDO DO_CLOSE_GR;
                MoveL Home_R_CW,v150,fine,Servo;
                PulseDO DO_OPEN_GR;
                WaitTime 0.25;
                PulseDO DO_DETACH_GR;
                WaitTime 0.25;
                MoveL Offs(Home_R_CW,0,30,0),v150,fine,Servo;
                MoveL Offs(Home_R,0,30,0),v150,fine,Servo;
                MoveL Home_R,v150,fine,Servo;
!                HOME;
                PulseDO DO_CLOSE_GR;
                WaitTime 0.25;
                PulseDO DO_ATTACH_4_GR;
                WaitTime 0.25;
!                SetDO DO_L_in_pos,1;
!                WaitDI DI_R_in_pos,0;
!                SetDO DO_L_in_pos,0;
            CASE "D" :      !cekej signal####################
                WaitDI DI_R_in_pos,1;
                PulseDO DO_OPEN_GR;
                WaitTime 0.25;
                PulseDO DO_DETACH_GR;
                WaitTime 0.25;
                HOME_DOWN;
                PulseDO DO_CLOSE_GR;
                WaitTime 0.25;
                PulseDO DO_ATTACH_3_GR;
                WaitTime 0.25;
                MoveL Offs(R_down_CW,0,0,-3),v150,fine,Servo;
                PulseDO DO_OPEN_GR;
                WaitTime 0.25;
                PulseDO DO_DETACH_GR;
                WaitTime 0.25;
                MoveL Offs(R_down_CW,0,0,-26),v150,fine,Servo;
                MoveL Offs(R_down,0,0,-26),v150,fine,Servo;
                MoveL Offs(R_down,0,0,-3),v150,fine,Servo;
                DOWN_HOME;
                PulseDO DO_CLOSE_GR;
                WaitTime 0.25;
                PulseDO DO_ATTACH_4_GR;
                WaitTime 0.25;
                SetDO DO_L_in_pos,1;
                WaitDI DI_R_in_pos,0;
                SetDO DO_L_in_pos,0;
            CASE "U2" :
                PulseDO DO_OPEN_GR;
                WaitTime 0.25;
                PulseDO DO_DETACH_GR;
                WaitTime 0.25;
                HOME_DOWN;
                PulseDO DO_CLOSE_GR;
                WaitTime 0.25;
                PulseDO DO_ATTACH_3_GR;
                WaitTime 0.25;
                SetDO DO_L_in_pos,1;
                WaitDI DI_R_in_pos,1;
                PulseDO DO_OPEN_GR;
                WaitTime 0.25;
                PulseDO DO_DETACH_GR;
                WaitTime 0.25;
                DOWN_HOME;
                PulseDO DO_CLOSE_GR;
                WaitTime 0.25;
                PulseDO DO_ATTACH_4_GR;
                WaitTime 0.25;
                SetDO DO_L_in_pos,0;
            CASE "F2" :
                PulseDO DO_OPEN_GR;
                WaitTime 0.25;
                PulseDO DO_DETACH_GR;
                WaitTime 0.25;
                HOME_BACK;
                PulseDO DO_CLOSE_GR;
                WaitTime 0.25;
                PulseDO DO_ATTACH_5_GR;
                WaitTime 0.25;
                SetDO DO_L_in_pos,1;
                WaitDI DI_R_in_pos,1;
                PulseDO DO_OPEN_GR;
                WaitTime 0.25;
                PulseDO DO_DETACH_GR;
                WaitTime 0.25;
                BACK_HOME;
                PulseDO DO_CLOSE_GR;
                WaitTime 0.25;
                PulseDO DO_ATTACH_4_GR;
                WaitTime 0.25;
                SetDO DO_L_in_pos,0;
            CASE "B2" :
                WaitDI DI_R_in_pos,1;
                PulseDO DO_OPEN_GR;
                WaitTime 0.25;
                PulseDO DO_DETACH_GR;
                WaitTime 0.25;
                HOME_BACK;
                PulseDO DO_CLOSE_GR;
                WaitTime 0.25;
                PulseDO DO_ATTACH_5_GR;
                WaitTime 0.25;
                MoveL R_back_CW,v150,fine,Servo;
                PulseDO DO_OPEN_GR;
                WaitTime 0.25;
                PulseDO DO_DETACH_GR;
                WaitTime 0.25;
                MoveL Offs(R_back_CW,-30,0,0),v150,fine,Servo;
                MoveL Offs(R_back,-30,0,0),v150,fine,Servo;
                MoveL R_back,v150,fine,Servo;
                PulseDO DO_CLOSE_GR;
                WaitTime 0.25;
                PulseDO DO_ATTACH_5_GR;
                WaitTime 0.25;
                MoveL R_back_CW,v150,fine,Servo;
                PulseDO DO_OPEN_GR;
                WaitTime 0.25;
                PulseDO DO_DETACH_GR;
                WaitTime 0.25;
                MoveL Offs(R_back_CW,-30,0,0),v150,fine,Servo;
                MoveL Offs(R_back,-30,0,0),v150,fine,Servo;
                MoveL R_back,v150,fine,Servo;
                BACK_HOME;
                PulseDO DO_CLOSE_GR;
                WaitTime 0.25;
                PulseDO DO_ATTACH_4_GR;
                WaitTime 0.25;
                SetDO DO_L_in_pos,1;
                WaitDI DI_R_in_pos,0;
                SetDO DO_L_in_pos,0;
            CASE "L2" :
!                PulseDO DO_OPEN_GR;
!                HOME;
!                PulseDO DO_CLOSE_GR;
!                SetDO DO_L_in_pos,1;
!                WaitDI DI_R_in_pos,1;
!                PulseDO DO_OPEN_GR;
!                HOME;
!                PulseDO DO_CLOSE_GR;
!                SetDO DO_L_in_pos,0;
            CASE "R2" :
!                WaitDI DI_R_in_pos,1;
!                PulseDO DO_OPEN_GR;
!                HOME;
!                PulseDO DO_CLOSE_GR;
                MoveL Home_R_CW,v150,fine,Servo;
                PulseDO DO_OPEN_GR;
                WaitTime 0.25;
                PulseDO DO_DETACH_GR;
                WaitTime 0.25;
                MoveL Offs(Home_R_CW,0,30,0),v150,fine,Servo;
                MoveL Offs(Home_R,0,30,0),v150,fine,Servo;
                MoveL Home_R,v150,fine,Servo;
!                HOME;
                PulseDO DO_CLOSE_GR;
                WaitTime 0.25;
                PulseDO DO_ATTACH_4_GR;
                WaitTime 0.25;
                MoveL Home_R_CW,v150,fine,Servo;
                PulseDO DO_OPEN_GR;
                WaitTime 0.25;
                PulseDO DO_DETACH_GR;
                WaitTime 0.25;
                MoveL Offs(Home_R_CW,0,30,0),v150,fine,Servo;
                MoveL Offs(Home_R,0,30,0),v150,fine,Servo;
                MoveL Home_R,v150,fine,Servo;
!                HOME;
                PulseDO DO_CLOSE_GR;
                WaitTime 0.25;
                PulseDO DO_ATTACH_4_GR;
                WaitTime 0.25;
!                SetDO DO_L_in_pos,1;
!                WaitDI DI_R_in_pos,0;
!                SetDO DO_L_in_pos,0;
            CASE "D2" :
                WaitDI DI_R_in_pos,1;
                PulseDO DO_OPEN_GR;
                WaitTime 0.25;
                PulseDO DO_DETACH_GR;
                WaitTime 0.25;
                HOME_DOWN;
                PulseDO DO_CLOSE_GR;
                WaitTime 0.25;
                PulseDO DO_ATTACH_3_GR;
                WaitTime 0.25;
                MoveL Offs(R_down_CW,0,0,-3),v150,fine,Servo;
                PulseDO DO_OPEN_GR;
                WaitTime 0.25;
                PulseDO DO_DETACH_GR;
                WaitTime 0.25;
                MoveL Offs(R_down_CW,0,0,-26),v150,fine,Servo;
                MoveL Offs(R_down,0,0,-26),v150,fine,Servo;
                MoveL Offs(R_down,0,0,-3),v150,fine,Servo;
                PulseDO DO_CLOSE_GR;
                WaitTime 0.25;
                PulseDO DO_ATTACH_3_GR;
                WaitTime 0.25;
                MoveL Offs(R_down_CW,0,0,-3),v150,fine,Servo;
                PulseDO DO_OPEN_GR;
                WaitTime 0.25;
                PulseDO DO_DETACH_GR;
                WaitTime 0.25;
                MoveL Offs(R_down_CW,0,0,-26),v150,fine,Servo;
                MoveL Offs(R_down,0,0,-26),v150,fine,Servo;
                MoveL Offs(R_down,0,0,-3),v150,fine,Servo;
                DOWN_HOME;
                PulseDO DO_CLOSE_GR;
                WaitTime 0.25;
                PulseDO DO_ATTACH_4_GR;
                WaitTime 0.25;
                SetDO DO_L_in_pos,1;
                WaitDI DI_R_in_pos,0;
                SetDO DO_L_in_pos,0;
            CASE "U'" :
                PulseDO DO_OPEN_GR;
                WaitTime 0.25;
                PulseDO DO_DETACH_GR;
                WaitTime 0.25;
                HOME_DOWN;
                PulseDO DO_CLOSE_GR;
                WaitTime 0.25;
                PulseDO DO_ATTACH_3_GR;
                WaitTime 0.25;
                SetDO DO_L_in_pos,1;
                WaitDI DI_R_in_pos,1;
                PulseDO DO_OPEN_GR;
                WaitTime 0.25;
                PulseDO DO_DETACH_GR;
                WaitTime 0.25;
                DOWN_HOME;
                PulseDO DO_CLOSE_GR;
                WaitTime 0.25;
                PulseDO DO_ATTACH_4_GR;
                WaitTime 0.25;
                SetDO DO_L_in_pos,0;
            CASE "F'" :
                PulseDO DO_OPEN_GR;
                WaitTime 0.25;
                PulseDO DO_DETACH_GR;
                WaitTime 0.25;
                HOME_BACK;
                PulseDO DO_CLOSE_GR;
                WaitTime 0.25;
                PulseDO DO_ATTACH_5_GR;
                WaitTime 0.25;
                SetDO DO_L_in_pos,1;
                WaitDI DI_R_in_pos,1;
                PulseDO DO_OPEN_GR;
                WaitTime 0.25;
                PulseDO DO_DETACH_GR;
                WaitTime 0.25;
                BACK_HOME;
                PulseDO DO_CLOSE_GR;
                WaitTime 0.25;
                PulseDO DO_ATTACH_4_GR;
                WaitTime 0.25;
                SetDO DO_L_in_pos,0;
            CASE "B'" :
                WaitDI DI_R_in_pos,1;
                PulseDO DO_OPEN_GR;
                WaitTime 0.25;
                PulseDO DO_DETACH_GR;
                WaitTime 0.25;
                HOME_BACK;
                PulseDO DO_CLOSE_GR;
                WaitTime 0.25;
                PulseDO DO_ATTACH_5_GR;
                WaitTime 0.25;
                MoveL R_back_ACW,v150,fine,Servo;
                PulseDO DO_OPEN_GR;
                WaitTime 0.25;
                PulseDO DO_DETACH_GR;
                WaitTime 0.25;
                MoveL Offs(R_back_ACW,-30,0,0),v150,fine,Servo;
                MoveL Offs(R_back,-30,0,0),v150,fine,Servo;
                MoveL R_back,v150,fine,Servo;
                BACK_HOME;
                PulseDO DO_CLOSE_GR;
                WaitTime 0.25;
                PulseDO DO_ATTACH_4_GR;
                WaitTime 0.25;
                SetDO DO_L_in_pos,1;
                WaitDI DI_R_in_pos,0;
                SetDO DO_L_in_pos,0;
            CASE "L'" :                 !NENENENEcekej signal####################   NEMELO BY BYT NIC POTREBA
!                PulseDO DO_OPEN_GR;
!                HOME;
!                PulseDO DO_CLOSE_GR;
!                SetDO DO_L_in_pos,1;
!                WaitDI DI_R_in_pos,1;
!                PulseDO DO_OPEN_GR;
!                HOME;
!                PulseDO DO_CLOSE_GR;
!                SetDO DO_L_in_pos,0;
            CASE "R'" :
!                WaitDI DI_R_in_pos,1;
!                PulseDO DO_OPEN_GR;
!                HOME;
!                PulseDO DO_CLOSE_GR;
                MoveL Home_R_ACW,v150,fine,Servo;
                PulseDO DO_OPEN_GR;
                WaitTime 0.25;
                PulseDO DO_DETACH_GR;
                WaitTime 0.25;
                MoveL Offs(Home_R_ACW,0,30,0),v150,fine,Servo;
                MoveL Offs(Home_R,0,30,0),v150,fine,Servo;
                MoveL Home_R,v150,fine,Servo;
!                HOME;
                PulseDO DO_CLOSE_GR;
                WaitTime 0.25;
                PulseDO DO_ATTACH_4_GR;
                WaitTime 0.25;
!                SetDO DO_L_in_pos,1;
!                WaitDI DI_R_in_pos,0;
!                SetDO DO_L_in_pos,0;
            CASE "D'" :
                WaitDI DI_R_in_pos,1;
                PulseDO DO_OPEN_GR;
                WaitTime 0.25;
                PulseDO DO_DETACH_GR;
                WaitTime 0.25;
                HOME_DOWN;
                PulseDO DO_CLOSE_GR;
                WaitTime 0.25;
                PulseDO DO_ATTACH_3_GR;
                WaitTime 0.25;
                MoveL Offs(R_down_ACW,0,0,-3),v150,fine,Servo;
                PulseDO DO_OPEN_GR;
                WaitTime 0.25;
                PulseDO DO_DETACH_GR;
                WaitTime 0.25;
                MoveL Offs(R_down_ACW,0,0,-26),v150,fine,Servo;
                MoveL Offs(R_down,0,0,-26),v150,fine,Servo;
                MoveL Offs(R_down,0,0,-3),v150,fine,Servo;
                DOWN_HOME;
                PulseDO DO_CLOSE_GR;
                WaitTime 0.25;
                PulseDO DO_ATTACH_4_GR;
                WaitTime 0.25;
                SetDO DO_L_in_pos,1;
                WaitDI DI_R_in_pos,0;
                SetDO DO_L_in_pos,0;
            CASE "BREAK" :
                BREAK;
        ENDTEST

      ENDFOR

        !Add your code here
    ENDPROC

    PROC HOME_DOWN()
        MoveL Offs(Home_R,0,30,0),v150,fine,Servo;
        MoveL Offs(Home_R_help_down,0,30,-30),v150,fine,Servo;
        MoveL Offs(R_down_help,0,30,-26),v150,fine,Servo;
        MoveL Offs(R_down,0,0,-26),v150,fine,Servo;
        MoveL Offs(R_down,0,0,-3),v150,fine,Servo;
        !MoveL R_down,v150,fine,Servo;
    ENDPROC
    PROC From_Home_to_Down()
        MoveL Home_R,v150,fine,Servo\WObj:=wobj0;
        MoveL Home_R_help_down,v150,fine,Servo\WObj:=wobj0;
        MoveL R_down_help,v150,fine,Servo\WObj:=wobj0;
        MoveL R_down,v150,fine,Servo\WObj:=wobj0;
        MoveL R_down_ACW,v150,fine,Servo\WObj:=wobj0;
        MoveL R_down,v150,fine,Servo\WObj:=wobj0;
        MoveL R_down_CW,v150,fine,Servo\WObj:=wobj0;
        MoveL R_down,v150,fine,Servo\WObj:=wobj0;
    ENDPROC
    PROC DOWN_HOME()
        MoveL Offs(R_down,0,0,-10),v150,fine,Servo;
        MoveL Offs(R_down_help,0,30,-20),v150,fine,Servo;
        MoveL Offs(Home_R_help_down,0,30,-30),v150,fine,Servo;
        MoveL Offs(Home_R,0,30,0),v150,fine,Servo;
        MoveL Home_R,v150,fine,Servo;
    ENDPROC
    PROC Down_to_home()
        MoveL R_down,v150,fine,Servo\WObj:=wobj0;
        MoveL R_down_help,v150,fine,Servo\WObj:=wobj0;
        MoveL Home_R_help_down,v150,fine,Servo\WObj:=wobj0;
        MoveL Home_R,v150,fine,Servo\WObj:=wobj0;
        MoveL Home_R_CW,v150,fine,Servo\WObj:=wobj0;
        MoveJ Home_R,v150,fine,Servo\WObj:=wobj0;
        MoveL Home_R_ACW,v150,fine,Servo\WObj:=wobj0;
        MoveJ Home_R,v150,fine,Servo\WObj:=wobj0;
    ENDPROC
    PROC HOME_BACK()
        MoveL Offs(Home_R,0,30,0),v150,fine,Servo;
        MoveL Offs(Home_R_help_back,-30,30,0),v150,fine,Servo;
        MoveJ Offs(R_back_help,-30,30,0),v150,fine,Servo;
        MoveL Offs(R_back,-30,0,0),v150,fine,Servo;
        MoveL R_back,v150,fine,Servo;
    ENDPROC
    PROC From_home_to_back()
        MoveL Home_R,v150,fine,Servo\WObj:=wobj0;
        MoveL Home_R_help_back,v150,fine,Servo\WObj:=wobj0;
        MoveJ R_back_help,v150,fine,Servo\WObj:=wobj0;
        MoveL R_back,v150,fine,Servo\WObj:=wobj0;
        MoveL R_back_CW,v150,fine,Servo\WObj:=wobj0;
        MoveL R_back,v150,fine,Servo\WObj:=wobj0;
        MoveL R_back_ACW,v150,fine,Servo\WObj:=wobj0;
        MoveL R_back,v150,fine,Servo\WObj:=wobj0;
    ENDPROC
    PROC BACK_HOME()
        MoveL Offs(R_back,-30,0,0),v150,fine,Servo;
        MoveL Offs(R_back_help,-30,30,0),v150,fine,Servo;
        MoveJ Offs(Home_R_help_back,-30,30,0),v150,fine,Servo;
        MoveL Offs(Home_R,0,30,0),v150,fine,Servo;
        MoveL Home_R,v150,fine,Servo;
    ENDPROC
    PROC From_back_to_home()
        MoveL R_back,v150,fine,Servo\WObj:=wobj0;
        MoveL R_back_help,v150,fine,Servo\WObj:=wobj0;
        MoveJ Home_R_help_back,v150,fine,Servo\WObj:=wobj0;
        MoveL Home_R,v150,fine,Servo\WObj:=wobj0;
        MoveL Home_R_CW,v150,fine,Servo\WObj:=wobj0;
        MoveJ Home_R,v150,fine,Servo\WObj:=wobj0;
        MoveL Home_R_ACW,v150,fine,Servo\WObj:=wobj0;
        MoveJ Home_R,v150,fine,Servo\WObj:=wobj0;
    ENDPROC
    PROC HOME()
        MoveJ Offs(Home_R,0,300,0),v150,fine,Servo;
        MoveJ Offs(Home_R,0,30,0),v150,fine,Servo;
        MoveL Home_R,v150,fine,Servo;
    ENDPROC
    PROC R_HOME()
        MoveJ Home_R,v150,fine,Servo\WObj:=wobj0;
        MoveL Home_R_ACW,v150,fine,Servo\WObj:=wobj0;
        MoveJ Home_R,v150,fine,Servo\WObj:=wobj0;
        MoveL Home_R_CW,v150,fine,Servo\WObj:=wobj0;
        MoveJ Home_R,v150,fine,Servo\WObj:=wobj0;
    ENDPROC
ENDMODULE

--- Controller Data/Controller1/SYSPAR/EIO.cfg ---
EIO:CFG_1.0:6:1::
#
SYSSIG_IN:

      -Signal "Collision_Avoidance" -Action "CollAvoidance"
#
INDUSTRIAL_NETWORK:

      -Name "EtherNetIP" -Connection "Private Network"\
      -Label "EtherNet/IP Adapter Network"

      -Name "DeviceNet" -Label "DeviceNet Master/Slave Network" -Address "2"
#
EIO_CROSS:

      -Name "Cross_Signal_Lamp" -Res "Signal_Lamp" -Act1 "DRV1BRAKE"
#
EIO_SIGNAL_SAFELEVEL:

      -Name "FlangePowerSafeLevel" -ActionWhenStartup "Last"
#
DEVICENET_DEVICE:

      -Name "D652_10" -VendorName "ABB Robotics" -ProductName "24 VDC Unit"\
      -Address 10 -ProductCode 26 -DeviceType 7 -ConnectionType "COS"\
      -OutputSize 2 -InputSize 2
#
DEVICENET_INTERNAL_DEVICE:

      -Name "DN_Internal_Device" -VendorName "ABB Robotics"\
      -ProductName "DeviceNet Internal Slave Device"
#
ETHERNETIP_INTERNAL_DEVICE:

      -Name "EN_Internal_Device" -VendorName "ABB Robotics"\
      -ProductName "EtherNet/IP Internal Adapter Device"
#
EIO_SIGNAL:

      -Name "custom_DI_0" -SignalType "DI" -Device "D652_10" -DeviceMap "0"

      -Name "custom_DI_1" -SignalType "DI" -Device "D652_10" -DeviceMap "1"

      -Name "custom_DI_2" -SignalType "DI" -Device "D652_10" -DeviceMap "2"

      -Name "custom_DI_3" -SignalType "DI" -Device "D652_10" -DeviceMap "3"

      -Name "custom_DI_4" -SignalType "DI" -Device "D652_10" -DeviceMap "4"

      -Name "custom_DI_5" -SignalType "DI" -Device "D652_10" -DeviceMap "5"

      -Name "custom_DI_6" -SignalType "DI" -Device "D652_10" -DeviceMap "6"

      -Name "custom_DI_7" -SignalType "DI" -Device "D652_10" -DeviceMap "7"

      -Name "custom_DO_0" -SignalType "DO" -Device "D652_10" -DeviceMap "0"

      -Name "custom_DO_1" -SignalType "DO" -Device "D652_10" -DeviceMap "1"

      -Name "custom_DO_2" -SignalType "DO" -Device "D652_10" -DeviceMap "2"

      -Name "custom_DO_3" -SignalType "DO" -Device "D652_10" -DeviceMap "3"

      -Name "custom_DO_4" -SignalType "DO" -Device "D652_10" -DeviceMap "4"

      -Name "custom_DO_5" -SignalType "DO" -Device "D652_10" -DeviceMap "5"

      -Name "custom_DO_6" -SignalType "DO" -Device "D652_10" -DeviceMap "6"

      -Name "custom_DO_7" -SignalType "DO" -Device "D652_10" -DeviceMap "7"

      -Name "hall_sensor_joint_1" -SignalType "DI" -Device "D652_10"\
      -DeviceMap "8"

      -Name "hall_sensor_joint_2" -SignalType "DI" -Device "D652_10"\
      -DeviceMap "9"

      -Name "hall_sensor_joint_3" -SignalType "DI" -Device "D652_10"\
      -DeviceMap "11"

      -Name "hall_sensor_joint_4" -SignalType "DI" -Device "D652_10"\
      -DeviceMap "12"

      -Name "hall_sensor_joint_5" -SignalType "DI" -Device "D652_10"\
      -DeviceMap "13"

      -Name "hall_sensor_joint_6" -SignalType "DI" -Device "D652_10"\
      -DeviceMap "14"

      -Name "hall_sensor_joint_7" -SignalType "DI" -Device "D652_10"\
      -DeviceMap "10"

      -Name "hall_sensor_24V_ROB_R" -SignalType "DO" -Device "D652_10"\
      -DeviceMap "8"

      -Name "hall_sensor_24V_ROB_L" -SignalType "DO" -Device "D652_10"\
      -DeviceMap "9"

      -Name "flange_24V_ROB_R" -SignalType "DO" -Device "D652_10"\
      -DeviceMap "10" -SafeLevel "FlangePowerSafeLevel"

      -Name "flange_24V_ROB_L" -SignalType "DO" -Device "D652_10"\
      -DeviceMap "11" -SafeLevel "FlangePowerSafeLevel"

      -Name "Signal_Lamp" -SignalType "DO" -Device "D652_10" -DeviceMap "12"

      -Name "Collision_Avoidance" -SignalType "DO" -Access "All" -Default 1

      -Name "DO_OPEN_GL" -SignalType "DO"

      -Name "DO_CLOSE_GL" -SignalType "DO"

      -Name "DO_OPEN_GR" -SignalType "DO"

      -Name "DO_CLOSE_GR" -SignalType "DO"

      -Name "DO_ATTACH_1_GL" -SignalType "DO"

      -Name "DO_ATTACH_2_GL" -SignalType "DO"

      -Name "DO_DETACH_GL" -SignalType "DO"

      -Name "DO_ATTACH_3_GR" -SignalType "DO"

      -Name "DO_ATTACH_4_GR" -SignalType "DO"

      -Name "DO_DETACH_GR" -SignalType "DO"

      -Name "DO_RESET_ENV" -SignalType "DO"

      -Name "DO_ATTACH_6_GL" -SignalType "DO"

      -Name "DO_ATTACH_5_GR" -SignalType "DO"

      -Name "DI_L_in_pos" -SignalType "DI"

      -Name "DI_R_in_pos" -SignalType "DI"

      -Name "DO_L_in_pos" -SignalType "DO"

      -Name "DO_R_in_pos" -SignalType "DO"
